SUBAPPLICATION IOAbstractionDemo (* IO Abstraction Layer pattern demo: logiBUS_IE/logiBUS_QX as Hardware+HAL layers around the fully event-driven EventDrivenCylinder application layer *)
  (* Standard: 61499-2; Description: Copyright (c) 2026 Meisterschulen am Ostbahnhof This program and the accompanying materials are made available under the terms of the Eclipse Public License 2.0 which is available at https://www.eclipse.org/legal/epl-2.0/ SPDX-License-Identifier: EPL-2.0 *)
  (* Version 1.0, 2026-08-31, Franz Höpfinger, Meisterschulen am Ostbahnhof, IO Abstraction Layer design pattern (IEC 61499 primer course, Module 6, Valeriy Vyatkin, slide 63), demo application *)
  PACKAGE Meins::DesingPatterns::IOAbstractionPattern;
  IMPORT logiBUS::io::DI::logiBUS_DI::Input_I1;
  IMPORT logiBUS::io::DI::logiBUS_DI::Input_I2;
  IMPORT logiBUS::io::DI::logiBUS_DI::Input_I3;
  IMPORT logiBUS::io::DI::logiBUS_DI::Input_I4;
  IMPORT logiBUS::io::DI::logiBUS_DI_Events::BUTTON_SINGLE_CLICK;
  IMPORT logiBUS::io::DQ::logiBUS_DO::Output_Q1;
  IMPORT logiBUS::io::DQ::logiBUS_DO::Output_Q2;
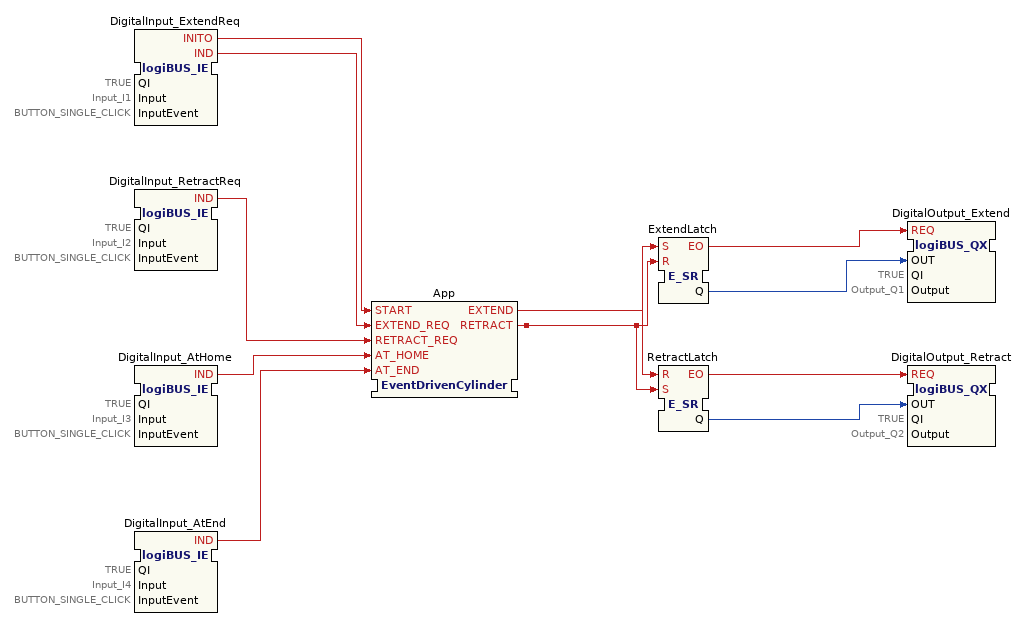
  FBS
    DigitalInput_ExtendReq : logiBUS::io::DI::logiBUS_IE(QI := TRUE, Input := Input_I1, InputEvent := BUTTON_SINGLE_CLICK);
    DigitalInput_RetractReq : logiBUS::io::DI::logiBUS_IE(QI := TRUE, Input := Input_I2, InputEvent := BUTTON_SINGLE_CLICK);
    DigitalInput_AtHome : logiBUS::io::DI::logiBUS_IE(QI := TRUE, Input := Input_I3, InputEvent := BUTTON_SINGLE_CLICK);
    DigitalInput_AtEnd : logiBUS::io::DI::logiBUS_IE(QI := TRUE, Input := Input_I4, InputEvent := BUTTON_SINGLE_CLICK);
    App : Meins::DesingPatterns::PurelyEventDrivenPattern::EventDrivenCylinder;
    ExtendLatch : iec61499::events::E_SR;
    RetractLatch : iec61499::events::E_SR;
    DigitalOutput_Extend : logiBUS::io::DQ::logiBUS_QX(QI := TRUE, Output := Output_Q1);
    DigitalOutput_Retract : logiBUS::io::DQ::logiBUS_QX(QI := TRUE, Output := Output_Q2);
  END_FBS
  EVENT_CONNECTIONS
    DigitalInput_ExtendReq.INITO TO App.START; (* Bootstrap: fires once at deployment *)
    DigitalInput_ExtendReq.IND TO App.EXTEND_REQ;
    DigitalInput_RetractReq.IND TO App.RETRACT_REQ;
    DigitalInput_AtHome.IND TO App.AT_HOME;
    DigitalInput_AtEnd.IND TO App.AT_END;
    App.EXTEND TO ExtendLatch.S;
    App.EXTEND TO RetractLatch.R;
    App.RETRACT TO RetractLatch.S;
    App.RETRACT TO ExtendLatch.R;
    ExtendLatch.EO TO DigitalOutput_Extend.REQ;
    RetractLatch.EO TO DigitalOutput_Retract.REQ;
  END_CONNECTIONS
  DATA_CONNECTIONS
    ExtendLatch.Q TO DigitalOutput_Extend.OUT;
    RetractLatch.Q TO DigitalOutput_Retract.OUT;
  END_CONNECTIONS
END_SUBAPPLICATION
